//{attribute 'conditionalshow' := 'SomeText'}
//{attribute 'conditionalshow'}
//{attribute 'hide'}
VAR_GLOBAL CONSTANT
END_VAR

(* stored: Version 1.1.0.1, ProductVersion 3.1.4024.12
   GVL Constants: Id {bff71fc4-b646-46ce-893a-6f98c40a3e79} *)
